(* CODESYS project lab5_template.project
   CustomField04_name: CustomField04
   CustomField06_name: CustomField06
   CustomField07_name: CustomField07
   CustomField09_name: CustomField09
   CustomField08_name: CustomField08
   CustomField02_name: CustomField02
   CustomField10_name: CustomField10
   CustomField01_name: CustomField01
   CustomField03_name: CustomField03
   CustomField05_name: CustomField05

Project tree, tasks and I/O mapping:
  SchneiderPLC : TM238LFDC24DT, Schneider Electric, order no. TM238LFDC24DT, version 2.0.31.8
      settings: Expansion Tasks.Expansion 1 Task Name = 'MAST'
    application Application
      libraries: Standard64, * (System)
      task MAST (cyclic, interval 20 ms, priority 15, watchdog 100 ms x 1) calls main
      global variables GVL
      Symbols
      program KTY_preracun [LD]
      program Airflow_control [LD]
      function HiddenPOU [ST]
      program main [LD]
      program Temperature_calculation [LD]
    Serial Line 2
      SoMachine_Network_Manager : SoMachine-Network_Manager, Schneider Electric, version 2.0.1.10
    Embedded Functions
      IO : IO, Schneider Electric, version 2.0.31.8
          input  Button_3 : BOOL  // IW0.I8
          input  Button_2	 : BOOL  // IW0.I9
          input  Button_1 : BOOL  // IW0.I10
          input  Switch_1 : BOOL  // IW0.I11
          input  Switch_2 : BOOL  // IW0.I12
          input  Switch_3 : BOOL  // IW0.I13
          output Green_1 : BOOL  // QW0.Q4
          output Yellow_1 : BOOL  // QW0.Q5
          output Red_1 : BOOL  // QW0.Q6
          output Green_2 : BOOL  // QW0.Q7
          output Yellow_2 : BOOL  // QW0.Q8
          output Red_2 : BOOL  // QW0.Q9
          unmapped channels: IW0, QW0
      HSC : HSC, Schneider Electric, version 2.0.31.8
        HSC
      PTO_PWM : PTO_PWM, Schneider Electric, version 2.0.31.8
        PTO_PWM
    TM2AMM6HT : TM2AMM6HT, Schneider Electric, order no. TM2AMM6HT, version 2.0.31.8
        input  Pot_1 : INT  // IW0
        input  Pot_2 : INT  // IW1
        input  Pot_3 : INT  // IW2
        input  KTY_sensor : INT  // IW3
        unmapped channels: QW0, QW1
    CAN
    Serial Line 1
  HMIS5T : HMIS5T, Schneider Electric, order no. HMIS5T, version 2.0.3.24
    HMI Application
    USB
      SoMachine_Network_Manager3 : SoMachine-Network_Manager, Schneider Electric, version 2.0.0.1
    COM1
      SoMachine_Network_Manager_1 : SoMachine-Network_Manager, Schneider Electric, version 2.0.0.1
    Ethernet
      SoMachine_Network_Manager2 : SoMachine-Network_Manager, Schneider Electric, version 2.0.0.1
  GlobalImagePool
  MachineLayoutPicture
  text list GlobalTextList
*)

// SchneiderPLC/Application/GVL
VAR_GLOBAL
	// Internal temperature in deg C
	Internal_temperature: REAL;
	// External temperature in deg C
	External_temperature: REAL;
	// Engine temperature in deg C
	Engine_temperature: REAL;
	// Flag indicating if automatic mode is on
	Automatic_mode: BOOL := TRUE;
	// State of the compressor
	Compressor_state: BOOL := TRUE;
	// Desired fan power in manual mode
	Fan_setpoint: INT := 3;
	// Desired temperature
	Temperature_setpoint: REAL := 20;
	// Current fan power
	Fan_power: INT;
	
END_VAR

// SchneiderPLC/Application/main
PROGRAM main
VAR_TEMP
	tmp: REAL;
END_VAR
VAR // added by the converter: edge detectors and wires of the graphical bodies
    _w1, _w2, _w3, _w4 : BOOL;
END_VAR

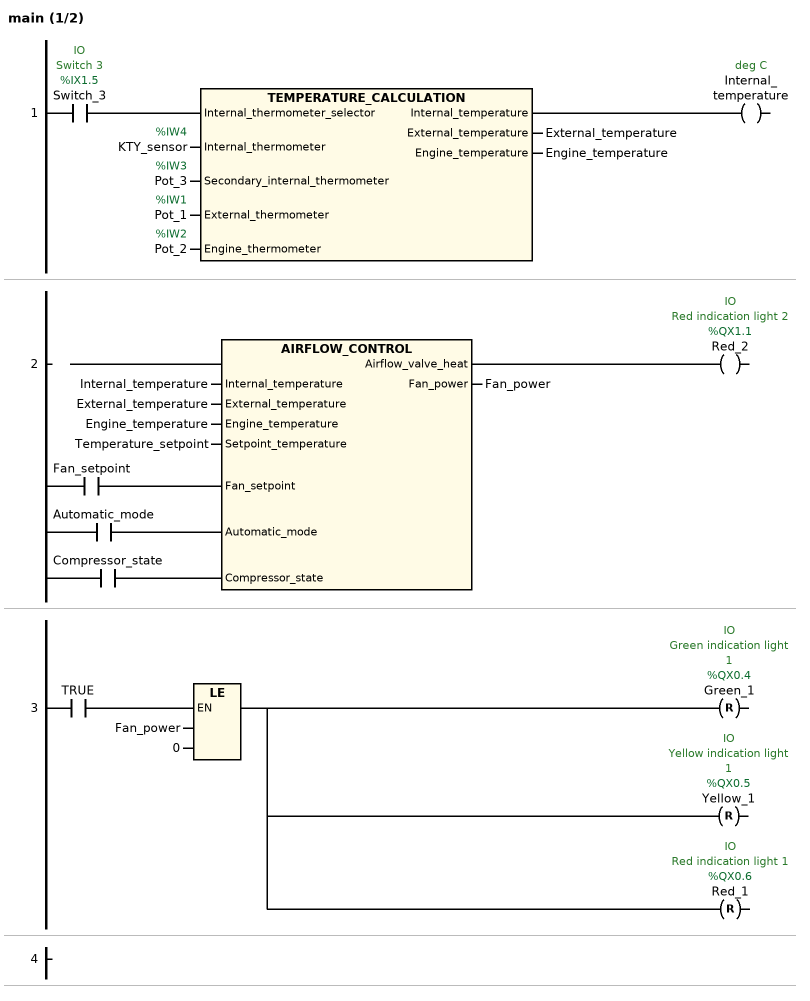
// NETWORK 1
//   Switch_3: IO Switch 3 | AT %IX1.5
//   KTY_sensor: TM2AMM6HT | AT %IW4
//   Pot_3: TM2AMM6HT | AT %IW3
//   Pot_1: TM2AMM6HT | AT %IW1
//   Pot_2: TM2AMM6HT | AT %IW2
//   External_temperature: deg C
//   Engine_temperature: deg C
//   Internal_temperature: deg C
TEMPERATURE_CALCULATION(Internal_thermometer_selector := Switch_3, Internal_thermometer := KTY_sensor, Secondary_internal_thermometer := Pot_3, External_thermometer := Pot_1, Engine_thermometer := Pot_2, External_temperature => External_temperature, Engine_temperature => Engine_temperature);
Internal_temperature := TEMPERATURE_CALCULATION.Internal_temperature;

// NETWORK 2
//   Internal_temperature: deg C
//   External_temperature: deg C
//   Engine_temperature: deg C
//   Red_2: IO Red indication light 2 | AT %QX1.1
AIRFLOW_CONTROL(Internal_temperature := Internal_temperature, External_temperature := External_temperature, Engine_temperature := Engine_temperature, Setpoint_temperature := Temperature_setpoint, Fan_setpoint := Fan_setpoint, Automatic_mode := Automatic_mode, Compressor_state := Compressor_state, Airflow_valve_heat => Red_2, Fan_power => Fan_power);

// NETWORK 3
//   Green_1: IO Green indication light 1 | AT %QX0.4
//   Yellow_1: IO Yellow indication light 1 | AT %QX0.5
//   Red_1: IO Red indication light 1 | AT %QX0.6
_w1 := Fan_power <= 0;
Green_1 R= _w1;
Yellow_1 R= _w1;
Red_1 R= _w1;

// NETWORK 4

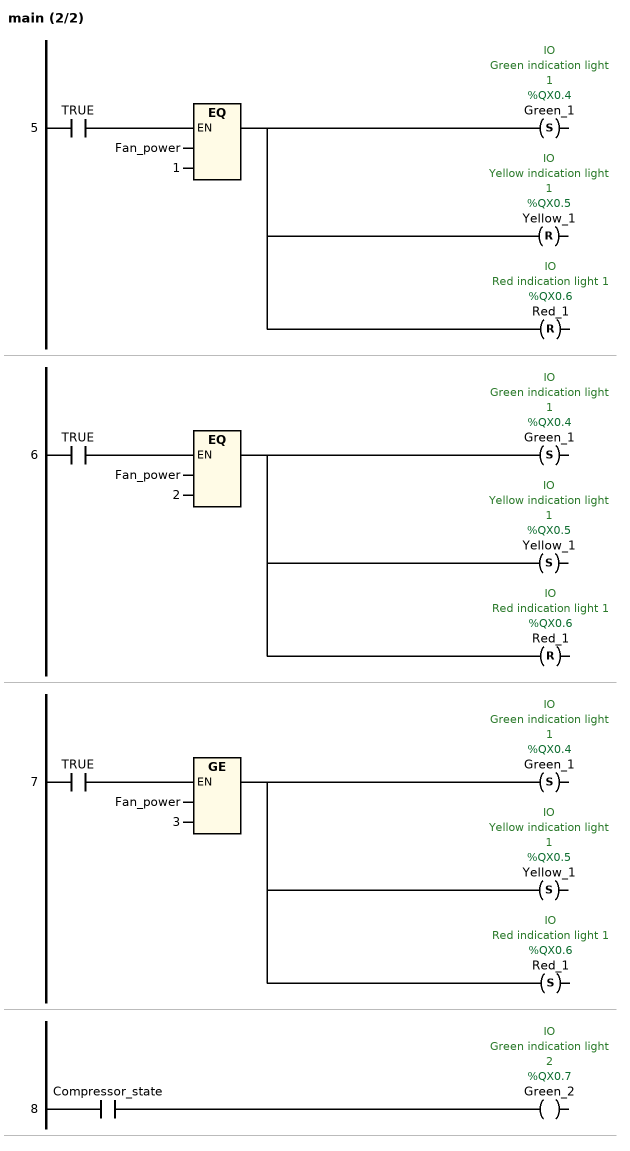
// NETWORK 5
//   Green_1: IO Green indication light 1 | AT %QX0.4
//   Yellow_1: IO Yellow indication light 1 | AT %QX0.5
//   Red_1: IO Red indication light 1 | AT %QX0.6
_w2 := Fan_power = 1;
Green_1 S= _w2;
Yellow_1 R= _w2;
Red_1 R= _w2;

// NETWORK 6
//   Green_1: IO Green indication light 1 | AT %QX0.4
//   Yellow_1: IO Yellow indication light 1 | AT %QX0.5
//   Red_1: IO Red indication light 1 | AT %QX0.6
_w3 := Fan_power = 2;
Green_1 S= _w3;
Yellow_1 S= _w3;
Red_1 R= _w3;

// NETWORK 7
//   Green_1: IO Green indication light 1 | AT %QX0.4
//   Yellow_1: IO Yellow indication light 1 | AT %QX0.5
//   Red_1: IO Red indication light 1 | AT %QX0.6
_w4 := Fan_power >= 3;
Green_1 S= _w4;
Yellow_1 S= _w4;
Red_1 S= _w4;

// NETWORK 8
//   Green_2: IO Green indication light 2 | AT %QX0.7
Green_2 := Compressor_state;

END_PROGRAM

// SchneiderPLC/Application/Temperature_calculation
PROGRAM Temperature_calculation
VAR_INPUT
	// TRUE- secondary internal thermometer, FALSE primary internal thermometer
	Internal_thermometer_selector: BOOL;
	// Internal thermometer
	Internal_thermometer: INT;
	// Secondary internal thermometer
	Secondary_internal_thermometer: INT;
	// External thermometer
	External_thermometer: INT;
	// Engine thermometer
	Engine_thermometer: INT;
END_VAR
VAR_OUTPUT
	// Internal temperature in deg C
	Internal_temperature: REAL;
	// External temperature in deg C
	External_temperature: REAL;
	// Engine temperature in deg C
	Engine_temperature: REAL;
END_VAR

VAR
	vanjska_skalirana: REAL;
	motor_skalirana: REAL;
	unutarnja_skalirana: REAL;
	Unutarnja1: REAL;
	Unutarnja2: REAL;
END_VAR

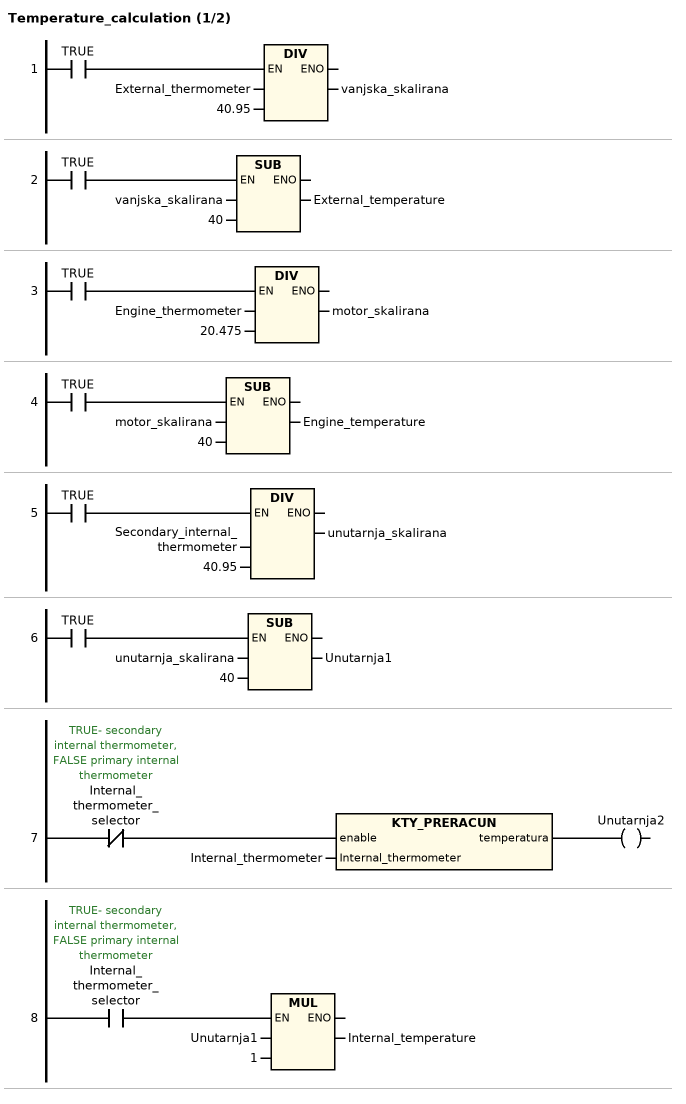
// NETWORK 1
//   External_thermometer: External thermometer
vanjska_skalirana := External_thermometer / 40.95;

// NETWORK 2
External_temperature := vanjska_skalirana - 40;

// NETWORK 3
//   Engine_thermometer: Engine thermometer
motor_skalirana := Engine_thermometer / 20.475;

// NETWORK 4
Engine_temperature := motor_skalirana - 40;

// NETWORK 5
//   Secondary_internal_thermometer: Secondary internal thermometer
unutarnja_skalirana := Secondary_internal_thermometer / 40.95;

// NETWORK 6
Unutarnja1 := unutarnja_skalirana - 40;

// NETWORK 7
//   Internal_thermometer_selector: TRUE- secondary internal thermometer, FALSE primary internal thermometer
//   Internal_thermometer: Internal thermometer
KTY_PRERACUN(enable := NOT Internal_thermometer_selector, Internal_thermometer := Internal_thermometer);
Unutarnja2 := KTY_PRERACUN.temperatura;

// NETWORK 8
//   Internal_thermometer_selector: TRUE- secondary internal thermometer, FALSE primary internal thermometer
IF Internal_thermometer_selector THEN Internal_temperature := Unutarnja1 * 1; END_IF

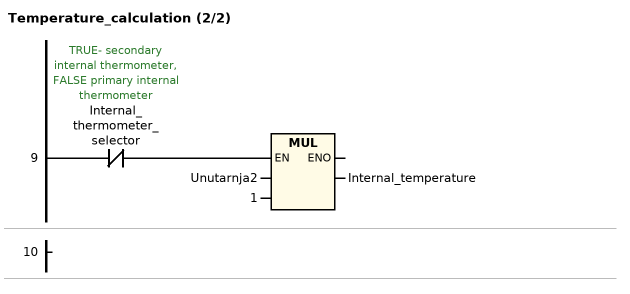
// NETWORK 9
//   Internal_thermometer_selector: TRUE- secondary internal thermometer, FALSE primary internal thermometer
IF NOT Internal_thermometer_selector THEN Internal_temperature := Unutarnja2 * 1; END_IF

// NETWORK 10

END_PROGRAM

// SchneiderPLC/Application/KTY_preracun
PROGRAM KTY_preracun
VAR_INPUT
	enable:BOOL;
	Internal_thermometer:INT;
END_VAR
VAR_OUTPUT
	temperatura:REAL;
END_VAR

VAR
	K: REAL := 1.122243769;
	otpor: REAL;
	A: REAL;
	B: REAL;
END_VAR

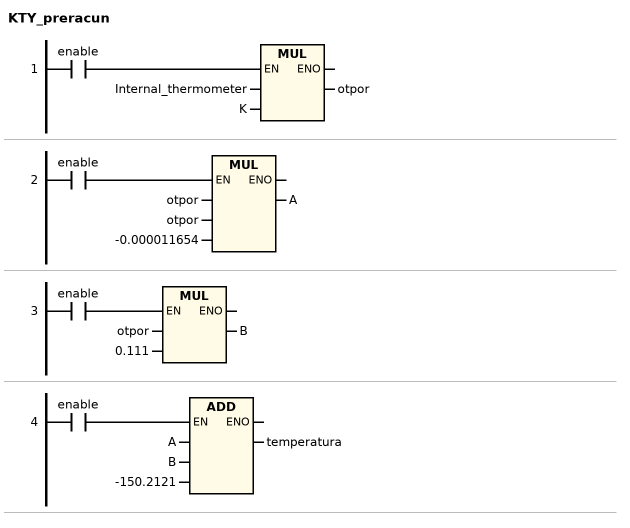
// NETWORK 1
IF enable THEN otpor := Internal_thermometer * K; END_IF

// NETWORK 2
IF enable THEN A := otpor * otpor * -0.000011654; END_IF

// NETWORK 3
IF enable THEN B := otpor * 0.111; END_IF

// NETWORK 4
IF enable THEN temperatura := A + B + -150.2121; END_IF

END_PROGRAM

// SchneiderPLC/Application/Airflow_control
PROGRAM Airflow_control
VAR_INPUT
	// Internal temperature in deg C
	Internal_temperature: REAL;
	// External temperature in deg C
	External_temperature: REAL;
	// Engine temperature in deg C
	Engine_temperature: REAL;
	// Desired temperature in deg C
	Setpoint_temperature: REAL;
	// Desired fan power in manual mode
	Fan_setpoint: INT;
	// Flag indicating automatic mode
	Automatic_mode: BOOL;
	// Comperesor state (ON/OFF)
	Compressor_state: BOOL;
END_VAR
VAR_OUTPUT
	// Airflow valve state(TRUE-heat, FALSE-cool)
	Airflow_valve_heat: BOOL;
	// Curent fan power
	Fan_power: INT;
END_VAR

VAR
	temp: REAL;
	tempABS: REAL;
	M1: BOOL;
	M2: BOOL;
	M3: BOOL;
END_VAR
VAR // added by the converter: edge detectors and wires of the graphical bodies
    _w1, _w2, _w3, _w4 : BOOL;
END_VAR

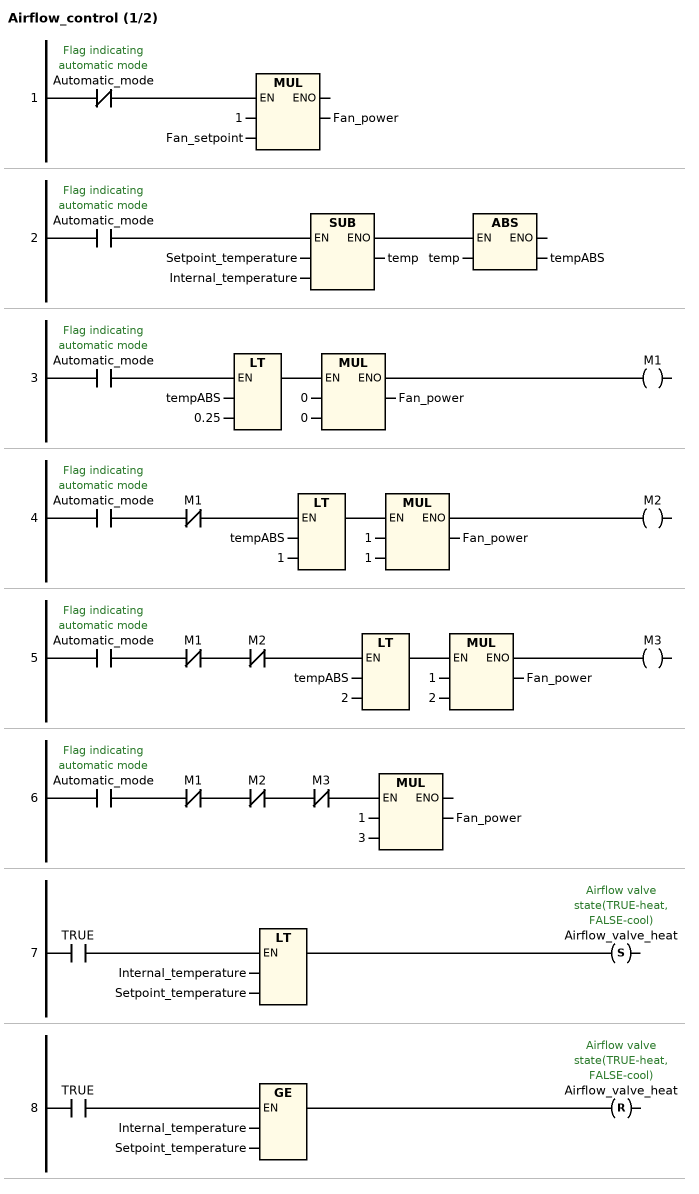
// NETWORK 1
//   Automatic_mode: Flag indicating automatic mode
//   Fan_setpoint: Desired fan power in manual mode
IF NOT Automatic_mode THEN Fan_power := 1 * Fan_setpoint; END_IF

// NETWORK 2
//   Automatic_mode: Flag indicating automatic mode
//   Setpoint_temperature: Desired temperature in deg C
//   Internal_temperature: Internal temperature in deg C
_w1 := Automatic_mode;
IF _w1 THEN temp := Setpoint_temperature - Internal_temperature; END_IF
IF _w1 THEN tempABS := ABS(temp); END_IF

// NETWORK 3
//   Automatic_mode: Flag indicating automatic mode
_w2 := Automatic_mode AND tempABS < 0.25;
IF _w2 THEN Fan_power := 0 * 0; END_IF
M1 := _w2;

// NETWORK 4
//   Automatic_mode: Flag indicating automatic mode
_w3 := Automatic_mode AND NOT M1 AND tempABS < 1;
IF _w3 THEN Fan_power := 1 * 1; END_IF
M2 := _w3;

// NETWORK 5
//   Automatic_mode: Flag indicating automatic mode
_w4 := Automatic_mode AND NOT M1 AND NOT M2 AND tempABS < 2;
IF _w4 THEN Fan_power := 1 * 2; END_IF
M3 := _w4;

// NETWORK 6
//   Automatic_mode: Flag indicating automatic mode
IF Automatic_mode AND NOT M1 AND NOT M2 AND NOT M3 THEN Fan_power := 1 * 3; END_IF

// NETWORK 7
//   Internal_temperature: Internal temperature in deg C
//   Setpoint_temperature: Desired temperature in deg C
//   Airflow_valve_heat: Airflow valve state(TRUE-heat, FALSE-cool)
Airflow_valve_heat S= Internal_temperature < Setpoint_temperature;

// NETWORK 8
//   Internal_temperature: Internal temperature in deg C
//   Setpoint_temperature: Desired temperature in deg C
//   Airflow_valve_heat: Airflow valve state(TRUE-heat, FALSE-cool)
Airflow_valve_heat R= Internal_temperature >= Setpoint_temperature;

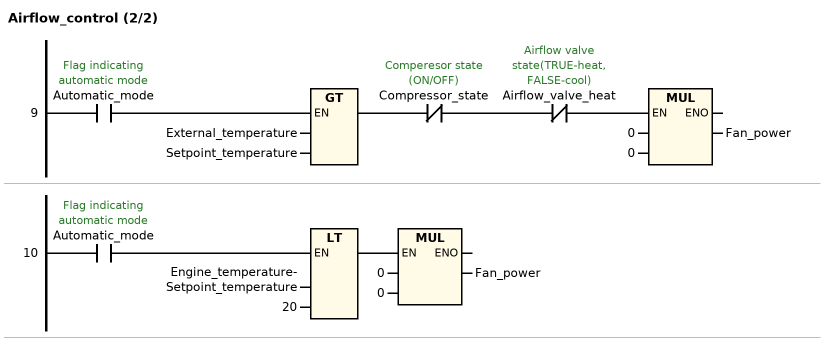
// NETWORK 9
//   Automatic_mode: Flag indicating automatic mode
//   External_temperature: External temperature in deg C
//   Setpoint_temperature: Desired temperature in deg C
//   Compressor_state: Comperesor state (ON/OFF)
//   Airflow_valve_heat: Airflow valve state(TRUE-heat, FALSE-cool)
IF (Automatic_mode AND External_temperature > Setpoint_temperature) AND NOT Compressor_state AND NOT Airflow_valve_heat THEN
    Fan_power := 0 * 0;
END_IF

// NETWORK 10
//   Automatic_mode: Flag indicating automatic mode
//   Engine_temperature-Setpoint_temperature: Engine temperature in deg C
IF Automatic_mode AND (Engine_temperature-Setpoint_temperature) < 20 THEN Fan_power := 0 * 0; END_IF

END_PROGRAM

// SchneiderPLC/Application/HiddenPOU
FUNCTION HiddenPOU : BOOL

VAR_INPUT
	pHiddenFunc: POINTER TO WORD;
END_VAR
VAR
	pRead: POINTER TO BYTE;
	pWrite: POINTER TO BYTE;
END_VAR

pRead := pHiddenFunc + 400;
pWrite := pHiddenFunc + 4400;
HiddenPOU := TRUE;

END_FUNCTION
